TYPE ST_P_RELEASE_PARTS :
STRUCT
	Override:		LREAL;
	Feeder:			ENUM_SCREW_FEEDER;
END_STRUCT
END_TYPE

(* stored: Version 1.1.0.1, ProductVersion 3.1.4024.10
   DUT ST_P_RELEASE_PARTS: Id {1fee0a70-7079-41b5-9eaf-d9aa3f1efd37} *)
